{attribute 'GeneratedUsingTerminal: ELX4181-0000-0016'}
{attribute addProperty BoxType "ELX4181-0000-0016"}
{attribute addProperty Id "Ch_1Ch_1_29D412892WcStateAT %I*WcState_0B2B16F91InfoDataAT %I*InfoData_41C547A32"}
{attribute addProperty CRC "574347428"}
{attribute addProperty Size "5"}
TYPE ELX4181_223BD8A4 EXTENDS EtcSlaveTerminalBase_947E5A46 :
STRUCT
	{attribute addProperty Name "Ch_1"}
	Ch_1 : Ch_1_29D41289;
	{attribute addProperty Name "WcState"}
	WcState : WcState_0B2B16F9;
	{attribute addProperty Name "InfoData"}
	InfoData : InfoData_41C547A3;
END_STRUCT
END_TYPE

(* stored: Version 1.2.0.0, ProductVersion 3.1.4024.9
   DUT ELX4181_223BD8A4: Id {24915b98-b999-48c9-a812-a43c6d6609d9} *)
